FUNCTION_BLOCK Seq_Set_MPlate EXTENDS FB_Basis IMPLEMENTS I_Sequenz
VAR_INPUT
	// Skillzuweisung
	R_Move			:I_Skill_RoboterErweitert;
	G_Move			:I_Skill_SmartGreifer; 
	
	// Prozessparameter		
	RobParam				:ARRAY[0..2] OF sRoboterProzessVariablen;
	GripParam				:sSmartGreiferProzessVariablen;
	ErreichtParam			:sKraftVariablen;
END_VAR
VAR_OUTPUT
END_VAR
VAR
	ErreichtParamReset		:sKraftVariablen;
END_VAR

// Ablauf
ACT_Ablauf();

// Zustandshandling
CASE iState OF
	0:	// BEREIT
		IF bStart THEN
			iState := 1;
		END_IF
	1:	// LAUFEND
		IF eSysCommand = 4 THEN
			bReset := TRUE;
			SFCReset := TRUE;
		END_IF
		
		IF bBeendet OR bReset THEN
			bReset := FALSE;
			SFCReset := FALSE;
			iState := 0;
		END_IF
	2: // ABGESCHLOSSEN
		IF SFCCurrentStep = 'Init' THEN
			iState := 0;
		END_IF
END_CASE

ACTION ACT_1:
R_Move.P_RobotParam := RobParam[0];
END_ACTION

ACTION ACT_2:
R_Move.P_RobotParam := RobParam[1];
R_Move.P_Erreicht := ErreichtParam;
END_ACTION

ACTION ACT_3:
G_Move.P_SGripperParam := GripParam;
END_ACTION

ACTION ACT_4:
R_Move.P_RobotParam := RobParam[2];
END_ACTION

ACTION ACT_Ablauf:
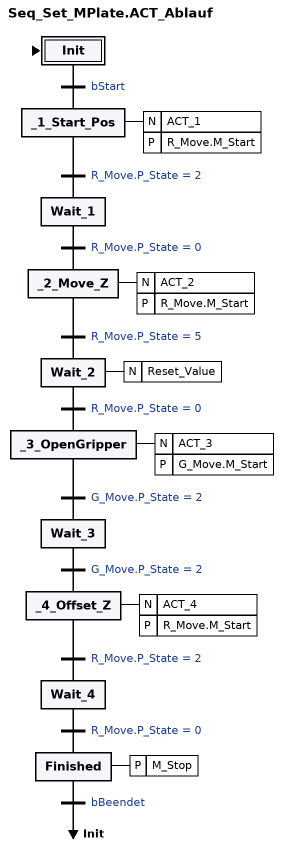
INITIAL_STEP Init:
END_STEP
TRANSITION FROM Init TO _1_Start_Pos
    := bStart;
END_TRANSITION
STEP _1_Start_Pos:
    ACT_1(N);
    R_Move.M_Start(P);
END_STEP
TRANSITION FROM _1_Start_Pos TO Wait_1
    := R_Move.P_State = 2;
END_TRANSITION
STEP Wait_1:
END_STEP
TRANSITION FROM Wait_1 TO _2_Move_Z
    := R_Move.P_State = 0;
END_TRANSITION
STEP _2_Move_Z:
    ACT_2(N);
    R_Move.M_Start(P);
END_STEP
TRANSITION FROM _2_Move_Z TO Wait_2
    := R_Move.P_State = 5;
END_TRANSITION
STEP Wait_2:
    Reset_Value(N);
END_STEP
TRANSITION FROM Wait_2 TO _3_OpenGripper
    := R_Move.P_State = 0;
END_TRANSITION
STEP _3_OpenGripper:
    ACT_3(N);
    G_Move.M_Start(P);
END_STEP
TRANSITION FROM _3_OpenGripper TO Wait_3
    := G_Move.P_State = 2;
END_TRANSITION
STEP Wait_3:
END_STEP
TRANSITION FROM Wait_3 TO _4_Offset_Z
    := G_Move.P_State = 2;
END_TRANSITION
STEP _4_Offset_Z:
    ACT_4(N);
    R_Move.M_Start(P);
END_STEP
TRANSITION FROM _4_Offset_Z TO Wait_4
    := R_Move.P_State = 2;
END_TRANSITION
STEP Wait_4:
END_STEP
TRANSITION FROM Wait_4 TO Finished
    := R_Move.P_State = 0;
END_TRANSITION
STEP Finished:
    M_Stop(P);
END_STEP
TRANSITION FROM Finished TO Init
    := bBeendet;
END_TRANSITION
END_ACTION

ACTION Reset_Value:
ErreichtParamReset.Fx := 0;
ErreichtParamReset.Fy := 0;
ErreichtParamReset.Fz := 0;

R_Move.P_Erreicht := ErreichtParamReset;
END_ACTION

END_FUNCTION_BLOCK

(* stored: Version 1.1.0.1
   POU Seq_Set_MPlate: Id {cafc47d7-0594-47cf-bec7-2bfe6cdf2092}, SpecialFunc None
   Folder 01_Zuweisung: Id {31a25897-d909-442b-a96e-55c02951eda5}
   Action ACT_1: Id {f8cb997d-1484-41a4-875a-7b624b127bf2}
   Action ACT_2: Id {f7277a6c-cb3c-4999-bfcc-87fa7dbf390c}
   Action ACT_3: Id {4bb91436-9d24-477a-a295-ef273ecbcadb}
   Action ACT_4: Id {f31313f6-0b4a-4866-bdc3-d481eff8a787}
   Action ACT_Ablauf: Id {f5d3ac2c-bc38-45bf-a603-c6ff0b029d61}
   Action Reset_Value: Id {3862e44f-e58a-468e-b2d7-a993f7feead8} *)
